PROGRAM MAIN
VAR
	Motor 					: ARRAY [1..4] OF FB_MOTOR;
	Simu 					: ARRAY [1..4] OF FB_SIM_MOTOR;
	sNames 					: ARRAY [1..4] OF STRING;
	State 					: ARRAY [1..4] OF States;
	previousState 			: ARRAY [1..4] OF States;
	bReset 			AT %I*	: ARRAY [1..4] OF BOOL;
	sMessage 		AT %I*	: ARRAY [1..4] OF STRING;
	bMove 			AT %I*	: ARRAY [1..4] OF BOOL;
	sMovType 		AT %I*	: ARRAY [1..4] OF STRING;
	lrPosition 		AT %I*	: ARRAY [1..4] OF LREAL;
	lrVelocity 		AT %I*	: ARRAY [1..4] OF LREAL;
	
	index					: INT;
	iNumber 				: INT;

	a: INT :=1;
	bStop: ARRAY [1..4] OF BOOL;
END_VAR

// Iniciamos los motores y sus simuladores
FOR index:=1 TO 4 DO
	sNames[index] := CONCAT('Motor', INT_TO_STRING(index));
	Motor[index](sName:=sNames[index], nNOVRAM_DevId:=0);
	Simu[index](ptrCfg:=ADR(Motor[index].cfg), ptrStat:=ADR(Motor[index].stat));
END_FOR

FOR iNumber := 1 TO 4 DO
	ACT_Mot();
END_FOR

//iNumber := 1;
//ACT_Mot();

ACTION ACT_Mot:
// Debido a que este código se basa en comandos RPC debemos poder parar su ejecución en cualquier momento
// si se activa el modo de control local
IF Motor[iNumber].stat.bLocal THEN
	previousState[iNumber] := State[iNumber];
	State[iNumber] := States.bLocal;
END_IF

IF bReset[iNumber] THEN
	State[iNumber] := States.Reset;
END_IF

CASE State[iNumber] OF
	
	States.bLocal :
		// Esperamos hasta que se desactiva el control local y volvemos al estado en el que nos encontrábamos.
		IF NOT Motor[iNumber].stat.bLocal THEN
			State[iNumber] := previousState[iNumber];
		END_IF
	
	States.Error :
		// En caso de error imprimimos el error en pantalla y esperamos a que el usuario nos de el OK para hacer un reset
		sMessage[iNumber] := CONCAT('Motor error: ', Motor[iNumber].stat.sErrorText);
		IF bReset[iNumber] THEN
			State[iNumber] := States.Reset;
		END_IF
		
	States.Stop :
		// En caso de solicitud de stop paramos el motor y volvemos al estado de espera de movimiento
		Motor[iNumber].RPC_Stop();
		State[iNumber] := States.MoveType;
		
	States.Reset :
		// Hacemos el reset y pasamos al estado de init
		Motor[iNumber].RPC_Reset();
		State[iNumber] := States.Init;
		bReset[iNumber] := FALSE;
	
	States.Init :
		// Ejecutamos el init y pasamos al estado de enable
		Motor[iNumber].RPC_Init();
		State[iNumber] := States.Enable;
		
	States.Enable :
		// Esperamos a que acabe la inicialización para realizar el enamble y pasar al siguiente estado
		IF Motor[iNumber].stat.bInitialised THEN
			Motor[iNumber].RPC_Enable();
			State[iNumber] := States.MoveType;
		// En caso de error durante el init pasamos al estado de reset
		ELSIF Motor[iNumber].stat.nStatus = E_MOTOR_STATUS.ERROR THEN
			State[iNumber] := States.Error;
		END_IF
		
	States.MoveType :
		// Comprobamos que no se haya producido ningún error en el movimiento anterior
		IF Motor[iNumber].stat.nStatus = E_MOTOR_STATUS.ERROR THEN
			State[iNumber] := States.Error;
		ELSE
			IF bStop[iNumber] THEN
				State[iNumber] := States.Stop;
				bStop[iNumber] := FALSE;
			// Esperamos a que el usuario active el movimiento para leer qué tipo de movimiento quiere hacer
			ELSIF bMove[iNumber] THEN
				bMove[iNumber] := FALSE;
				IF sMovType[iNumber] = 'Abs' THEN
					State[inumber] := States.Absolute;
					sMessage[iNumber] := '';             // En caso de que hubiese algún mensaje de tipo de movimiento erróneo anterior lo reseteamos
				ELSIF sMovType[iNumber] = 'Rel' THEN
					State[inumber] := States.Relative;
					sMessage[iNumber] := '';
				ELSIF sMovType[iNumber] = 'Vel' THEN
					State[inumber] := States.Velocity;
					sMessage[iNumber] := '';
				ELSE 
					sMessage[iNumber] := 'Wrong movement type input';
				END_IF
			END_IF
		END_IF
		
	States.Absolute :
		// Ejecutamos el movimiento absoluto
		Motor[iNumber].RPC_MoveAbs(in_lrPos := lrPosition[iNumber], in_lrVel := lrVelocity[iNumber]);
		State[iNumber] := States.MoveType;
		
	States.Relative :
		// Ejecutamos el movimiento relativo
		Motor[iNumber].RPC_MoveRel(in_lrPos := lrPosition[iNumber], in_lrVel := lrVelocity[iNumber]);
		State[iNumber] := States.MoveType;
		
	States.Velocity :
		// Ejecutamos el movimiento en velocidad
		Motor[iNumber].RPC_MoveVel(in_lrVel := lrVelocity[iNumber]);
		State[iNumber] := States.MoveType;
		
END_CASE
END_ACTION

END_PROGRAM

(* stored: Version 1.1.0.1, ProductVersion 3.1.4024.9
   POU MAIN: Id {86679b08-6d78-4646-b50c-b94e5d23f676}, SpecialFunc None
   Action ACT_Mot: Id {b8938c25-71e1-4140-baf5-76aca7db3f11} *)
